FUNCTION STR_TO_ASC : BYTE
VAR_INPUT
	str : STRING;
END_VAR
VAR
	pChar : POINTER TO BYTE;
END_VAR

	pChar 		:= ADR(str);
	STR_TO_ASC 	:= pChar^;

END_FUNCTION

(* stored: Version 1.1.0.1, ProductVersion 3.1.4024.16
   POU STR_TO_ASC: Id {eff02e5a-eb22-4acd-8922-0575f7d4a76e}, SpecialFunc None *)
